{attribute 'OPC.UA.DA.StructuredType' := '1'}
TYPE ST_SetPointState :
STRUCT
	fOperatingPoint	: REAL; //current operating point
	fSetPoint		: REAL; //current set point
	aSetPointLimits	: ARRAY[1..2] OF REAL; //lower and upper limit of setpoint
END_STRUCT
END_TYPE

(* stored: Version 1.1.0.1, ProductVersion 3.1.4024.9
   DUT ST_SetPointState: Id {a8ea9f16-1a3b-41a0-9776-e9b4f11e9876} *)
